// TIA Portal V20 export
VAR_GLOBAL   // PLC tag table "LGR_Const_Programs"
END_VAR
VAR_GLOBAL CONSTANT   // user constants
   TcpResQueMax : UInt := 100;
   EventQueMax : UInt := 100;
   PI : Real := 3.1415926535;
END_VAR
